TYPE ST_Setting :
STRUCT
	tPreSet 	: TIME; // Time to pass, before Q is set
END_STRUCT
END_TYPE

(* stored: Version 1.1.0.1, ProductVersion 3.1.4024.12
   DUT ST_Setting: Id {2eecb69a-08a0-4b01-b371-3f05ed33496c} *)
